(* PLC project KinIn_v3.project, CODESYS CODESYS V3.5 SP19 *)
(* stored: creationDateTime 2025-01-20T16:22:26.8299642, modificationDateTime 2025-01-20T16:17:39.6822999 *)

FUNCTION_BLOCK LuInverse
  VAR_INPUT
    {attribute 'variable_length_array_original_scope' := 'Inout'}
    {attribute 'variable_length_array' := 'ARRAY[*,*] OF REAL'}
    {attribute 'Dimensions' := '2'}
    L : POINTER TO REAL;
    {attribute 'variable_length_array_original_scope' := 'Inout'}
    {attribute 'variable_length_array' := 'ARRAY[*,*] OF REAL'}
    {attribute 'Dimensions' := '2'}
    u : POINTER TO REAL;
    {attribute 'variable_length_array_original_scope' := 'Inout'}
    {attribute 'variable_length_array' := 'ARRAY[*,*] OF REAL'}
    {attribute 'Dimensions' := '2'}
    a : POINTER TO REAL;
    {attribute 'variable_length_array_original_scope' := 'Inout'}
    {attribute 'variable_length_array' := 'ARRAY[*,*] OF REAL'}
    {attribute 'Dimensions' := '2'}
    d : POINTER TO REAL;
    {attribute 'variable_length_array_original_scope' := 'Inout'}
    {attribute 'variable_length_array' := 'ARRAY[*,*] OF REAL'}
    {attribute 'Dimensions' := '2'}
    eyeN : POINTER TO REAL;
  END_VAR
  VAR
    row : DINT;
    col : DINT;
    m : DINT;
    sumTemp_2 : REAL;
    sumTemp_d : REAL;
  END_VAR

            FOR col:=1 TO UPPER_BOUND(L,1) DO
    row:=1;
    for row:=1 TO UPPER_BOUND(L,1) DO
        //forward substitution
        m:=1;sumTemp_d:=0;
        for m:=1 TO row-1 DO
            sumTemp_d:=sumTemp_d+L[row,m]*d[m,col];
        end_for    
        d[row,col]:=eyeN[row,col]-sumTemp_d;
    end_for

    //backward substitution
    row:=UPPER_BOUND(L,1);
    FOR row:=UPPER_BOUND(L,1) TO 1 BY -1 DO
        m:=UPPER_BOUND(L,1);sumTemp_2:=0;
        FOR m:=UPPER_BOUND(L,1) TO row+1 BY -1 DO
            sumTemp_2:=sumTemp_2+u[row,m]*a[m,col];
        end_for    
        
		IF u[row,row]=0 AND (d[row,col]-sumTemp_2)=0 THEN
			a[row,col]:=1;
		ELSIF u[row,row]=0 THEN
			a[row,col]:=3.402823E+10;
		ELSE
			a[row,col]:=(d[row,col]-sumTemp_2)/u[row,row];
		END_IF
		
    end_for
end_for
          
END_FUNCTION_BLOCK
